FUNCTION_BLOCK EnumeratorConnection IMPLEMENTS I_EnumeratorConnection
VAR
	state : (VALID, INVALID) := VALID;
	updater : I_EnumeratorConnectionUpdater;
END_VAR

METHOD PUBLIC Dispose
VAR_INPUT
END_VAR
IF updater = 0 THEN
	RETURN;
END_IF

updater.RemoveConnection(this^);
END_METHOD

PROPERTY PUBLIC IsInvalid : BOOL
GET
IsInvalid := not IsValid;
END_GET
END_PROPERTY

PROPERTY PUBLIC IsValid : BOOL
GET
IsValid := state = VALID;
END_GET
END_PROPERTY

METHOD PUBLIC LinkTo
VAR_INPUT
	ConnectionUpdater : I_EnumeratorConnectionUpdater;
END_VAR
updater := ConnectionUpdater;
updater.AddConnection(this^);
END_METHOD

METHOD PUBLIC SetInvalid
VAR_INPUT
END_VAR
state := INVALID;
END_METHOD

METHOD PUBLIC SetValid
VAR_INPUT
END_VAR
state := VALID;
END_METHOD

END_FUNCTION_BLOCK

(* stored: Version 1.1.0.1, ProductVersion 3.1.4024.12
   POU EnumeratorConnection: Id {a89c3062-7404-4db8-85da-f08a8efbbeea}, SpecialFunc None
   Method Dispose: Id {c58b57c9-c08b-48b6-95a1-02c67bca0980}
   Property IsInvalid: Id {a16b766d-b64b-4d01-8d64-0a650e10d337}
   Get Get: Id {e1496e15-d5b0-482f-8d6e-5a47ac063db5}
   Property IsValid: Id {a308d4d3-7070-49c1-9e59-cb9afc7e166e}
   Get Get: Id {51c2e23f-46e4-42e2-81b3-9bc2d9115011}
   Method LinkTo: Id {132a622e-daae-470f-87ca-9d4c04618871}
   Method SetInvalid: Id {4fda179b-e030-441f-a8f0-0b0c361c4bf2}
   Method SetValid: Id {91e84979-b629-47b4-b564-6dd375674508} *)
